FUNCTION_BLOCK INTERNAL FINAL FB_ReadRepeatedFieldBytesTests EXTENDS FB_TestSuite
VAR_INPUT
END_VAR
VAR_OUTPUT
END_VAR
VAR
	aActual             : ARRAY[0..3] OF ARRAY[0..15] OF BYTE;
    fbFieldCodec 		: FB_FieldCodecBytes(nTag:= 16#22);
	fbRepeatedField		: FB_RepeatedField(anyArray:= F_ToAnyType(aActual), anyFirstElem:= F_ToAnyType(aActual[0]), ipFieldCodec:= fbFieldCodec);
END_VAR

ShouldReadRepeatedFieldTheory();

METHOD PRIVATE Reset
VAR_INPUT
END_VAR
fbRepeatedField.Initialize();
MEMSET(destAddr:= ADR(aActual), fillByte:= 16#0, n:= SIZEOF(aActual));
END_METHOD

METHOD PRIVATE ShouldReadRepeatedField
VAR_IN_OUT CONSTANT
    aBuffer     : ARRAY [*] OF BYTE;
    aExpected   : ARRAY[0..3] OF ARRAY[0..15] OF BYTE;
END_VAR
VAR_INPUT CONSTANT
    nBufferPosStart     : UDINT;
    nExpectedBufferPos  : UDINT;
    nExpectedFieldIndex : UDINT;
    ipFieldCodec        : I_FieldCodec;
END_VAR
VAR_INST
    fbCtx               : FB_ParseContext;
END_VAR
VAR
    hr                  : HRESULT;
    nTag                : UDINT;
    i                   : UDINT;
    aTmpBuffer          : ARRAY[0..1023] OF BYTE := [SIZEOF(aTmpBuffer)(16#FF)];
END_VAR
// Arrange
Reset();
fbCtx.FromBuffer(aBuffer);
fbCtx.refCtx.stState.nBufferPos := nBufferPosStart;
THIS^.fbFieldCodec.SetTmpBuffer(anyBytes:= F_ToAnyBytes(aTmpBuffer));

// Act
F_ParseTag(fbCtx.refCtx, nTag=> nTag);
hr := fbRepeatedField.AddEntriesFrom(fbParseCtx:= fbCtx, ipFieldCodec:= ipFieldCodec);

// Assert
AssertEquals_DINT(
    Expected:= S_OK,
    Actual:= hr,
    Message:= 'Expected S_OK instead of error');
    
{warning disable C0041}
FOR i:= 0 TO 3 DO
    AssertArrayEquals_BYTE(Expecteds:= aExpected[i], Actuals:= aActual[i], Message:= CONCAT('Array differs at index ', TO_STRING(i)));
END_FOR

AssertEquals_UDINT(
    Expected:= nExpectedBufferPos,
    Actual:= fbCtx.refCtx.stState.nBufferPos,
    Message:= CONCAT('Expected stState.nBufferPos to equal ', TO_STRING(nExpectedBufferPos)));
    
AssertEquals_UDINT(
    Expected:= nExpectedFieldIndex,
    Actual:= fbRepeatedField.nCount,
    Message:= CONCAT('Expected fbRepeatedField.nCount to equal ', TO_STRING(fbRepeatedField.nCount)));
END_METHOD

METHOD PRIVATE ShouldReadRepeatedFieldTheory : REFERENCE TO FB_Test
(*
    syntax = "proto3";
    
    message exampleMessage
    {
      repeated bytes repeatedBytes = 4;
    }    
*)

VAR CONSTANT
    cRawBytes1 : ARRAY[0..31] OF BYTE := [16#22, 16#03, 16#00, 16#01, 16#02, 16#22, 16#03, 16#03, 16#04, 16#05];
    
END_VAR

VAR CONSTANT
     aExpected1 : ARRAY[0..3] OF ARRAY[0..15] OF BYTE := [[0, 1, 2], [3, 4, 5]];
END_VAR
VAR
    // aBuffer     : ARRAY[0..1023] OF BYTE;       // tmp. buffer if chunks are larger then 256 bytes.
END_VAR
TEST(__POUNAME());

ShouldReadRepeatedField(aBuffer:= cRawBytes1, aExpected:= aExpected1, nBufferPosStart:= 0, nExpectedBufferPos:= 11, nExpectedFieldIndex:= 2, THIS^.fbFieldCodec);

TEST_FINISHED_NAMED(__POUNAME());
END_METHOD

END_FUNCTION_BLOCK

(* stored: Version 1.1.0.1
   POU FB_ReadRepeatedFieldBytesTests: Id {9d94c254-9f05-4fb3-94a3-cf2c4237a310}, SpecialFunc None
   Method Reset: Id {7e0c1d49-ab8c-4abf-b8a2-17987738c598}
   Method ShouldReadRepeatedField: Id {3988edba-b328-4893-819d-70d3231abe44}
   Method ShouldReadRepeatedFieldTheory: Id {5b11e0b5-8f5f-42bc-b128-9296078ae4aa} *)
